FUNCTION_BLOCK RASPBERRY_PI_GPIO_OUT
  {SET_ATTRIBUTE(OpcUa, DEVICE.SENSOR)}
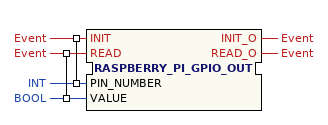
  EVENT_INPUT
    INIT WITH PIN_NUMBER;
    READ WITH VALUE;
  END_EVENT
  EVENT_OUTPUT
    INIT_O;
    READ_O;
  END_EVENT
  VAR_INPUT
    PIN_NUMBER : INT; {SET_ATTRIBUTE(OpcUa, Constant.RUN)}
    VALUE : BOOL; {SET_ATTRIBUTE(OpcUa, Variable.RUN)}
  END_VAR
END_FUNCTION_BLOCK
